INTERFACE I_Command EXTENDS I_Disposable

METHOD Execute
VAR_INPUT
END_VAR
END_METHOD

END_INTERFACE

(* stored: Version 1.1.0.1, ProductVersion 3.1.4024.12
   Itf I_Command: Id {8b8ba27f-662c-415c-9762-a176d8dd270a}
   Method Execute: Id {123bd7c2-e5d6-44cb-a05d-9fe45623507a} *)
